# EPICS substitutions: ek9000App/Db/EL1094.substitutions
file EL1094.template
{ 	pattern
	{
		TERMINAL,

	}
	{
	}
}
